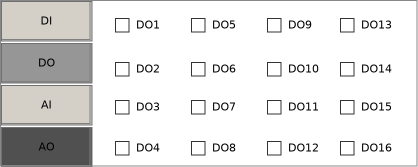
VISUALIZATION Digital_Outputs  // 418x167
    Button (1,127 91x40), "AO"
        OnMouseUp: change screen: Analog_Outputs
    Button (1,1 91x40), "DI"
        OnMouseUp: change screen: Digital_Inputs
    Button (1,43 91x40), "DO"
        OnMouseDown: change screen: Digital_Outputs
        OnMouseUp: change screen: Digital_Outputs
    Button (1,85 91x40), "AI"
        OnMouseUp: change screen: Analog_Inputs
    Checkbox (113,10 62x30), "DO1", variable: GVL_IO.DO1
    Checkbox (113,54 62x30), "DO2", variable: GVL_IO.DO2
    Checkbox (113,92 62x30), "DO3", variable: GVL_IO.DO3
    Checkbox (113,133 62x30), "DO4", variable: GVL_IO.DO4
    Checkbox (189,10 62x30), "DO5", variable: GVL_IO.DO5
    Checkbox (189,54 62x30), "DO6", variable: GVL_IO.DO6
    Checkbox (189,92 62x30), "DO7", variable: GVL_IO.DO7
    Checkbox (189,133 62x30), "DO8", variable: GVL_IO.DO8
    Checkbox (265,10 62x30), "DO9", variable: GVL_IO.DO9
    Checkbox (265,54 74x30), "DO10", variable: GVL_IO.DO10
    Checkbox (265,92 71x30), "DO11", variable: GVL_IO.DO11
    Checkbox (265,133 72x30), "DO12", variable: GVL_IO.DO12
    Checkbox (338,10 69x30), "DO13", variable: GVL_IO.DO13
    Checkbox (338,54 80x30), "DO14", variable: GVL_IO.DO14
    Checkbox (338,92 72x30), "DO15", variable: GVL_IO.DO15
    Checkbox (338,133 77x30), "DO16", variable: GVL_IO.DO16
END_VISUALIZATION

(* stored: Version 1.1.0.1, ProductVersion 3.1.4024.4
   Visu Digital_Outputs: Id {0d021015-0748-42b9-8585-df2155382b06} *)
